# EPICS autosave request: mtcaAnalyzerIOC/as/req/auto_settings.req
$(P)$(R)$(CH)Gain
$(P)$(R)$(CH)Offset
